PROGRAM PRG_KFE_RIX_VAC_FS
VAR
END_VAR

//Fast Shutter Valve

fb_TV1K2_VFS_1(
	i_xPMPS_OK:= TRUE, 
	i_xExt_OK:= TRUE, 
	i_sDevName:= 'TV1K2:VFS:1',
	io_fbFFHWO:= g_FastFaultOutput2
);
(*FastFaultOuput*)	
g_FastFaultOutput2.Execute(bAutoReset:= TRUE);

END_PROGRAM

(* stored: Version 1.1.0.1, ProductVersion 3.1.4024.2
   POU PRG_KFE_RIX_VAC_FS: Id {b788d1e6-f841-4e72-96a7-0fa8f5d54d8b}, SpecialFunc None *)
